{attribute 'linkalways'} 
{attribute 'no_explicit_call' := 'This FB is a CLASS and must be accessed using methods or properties'}
{attribute 'enable_dynamic_creation'}
FUNCTION_BLOCK _Array0to1_0to10OfBool EXTENDS ArrayDatatypeBase
VAR CONSTANT
	lBound : DINT := 0;
	uBound : DINT := 10;
END_VAR
VAR
	localData : ARRAY [0..1, 0..10] OF BOOL;
	activeData : REFERENCE TO ARRAY [0..1, 0..10] OF BOOL REF= localData;
	elements : ARRAY [0..1, 0..10] OF _BOOL(FALSE);
	elementLookup : Dictionary;
	baseType : _BOOL(FALSE);
END_VAR

PROPERTY PUBLIC Address : PVOID
GET
Address := ADR(activeData);
END_GET
END_PROPERTY

PROPERTY PUBLIC BaseDatatype : I_Datatype
GET
BaseDatatype := baseType;
END_GET
END_PROPERTY

METHOD PUBLIC ClearReference
VAR_INPUT
END_VAR
activeData REF= localData;
SetElementReference();
END_METHOD

METHOD PUBLIC Clone : I_Datatype
VAR
    pClone : POINTER TO _Array0to10OfBool;
END_VAR
pClone := __NEW(_Array0to10OfBool());
pClone^.Value := Value;
Clone := pClone^;
END_METHOD

METHOD FB_init : BOOL
VAR_INPUT
	bInitRetains : BOOL; // if TRUE, the retain variables are initialized (warm start / cold start)
	bInCopyCode : BOOL;  // if TRUE, the instance afterwards gets moved into the copy code (online change)
END_VAR
StoreElementsInLookup();
SetElementReference();
END_METHOD

METHOD PUBLIC GetElementAsDatatypeByIndex : I_Datatype
VAR_INPUT
	Index : DINT;
END_VAR
GetElementAsDatatypeByIndex := elements[Index];
END_METHOD

METHOD PUBLIC GetElementByIndex : REFERENCE TO _BOOL;
VAR_INPUT
	Index : DINT;
END_VAR
GetElementByIndex REF= elements[Index];
END_METHOD

PROPERTY PUBLIC LowerBound : DINT
GET
LowerBound := lBound;
END_GET
END_PROPERTY

METHOD PUBLIC MakeReferenceTo
VAR_INPUT
	ReferenceTarget : REFERENCE TO ARRAY [lBound..uBound] OF BOOL;
END_VAR
activeData REF= ReferenceTarget;
SetElementReference();
END_METHOD

METHOD PROTECTED OnSerializeArrayValues
VAR_INPUT
	Serializer : I_Serializer;
END_VAR
VAR
	i : DINT;
END_VAR
FOR i := lBound TO uBound DO
	elements[i].SerializeWith(Serializer);
END_FOR
END_METHOD

METHOD PROTECTED SetElementReference
VAR_INPUT
END_VAR
VAR
	i : DINT;
END_VAR
FOR i := lBound TO uBound DO
	elements[i].MakeReferenceTo(activeData[i]);
END_FOR
END_METHOD

PROPERTY PUBLIC Size : UDINT
GET
Size := SIZEOF(activeData);
END_GET
END_PROPERTY

METHOD PROTECTED StoreElementsInLookup
VAR_INPUT
END_VAR
FOR i := lBound TO uBound DO
	elements[i].MakeReferenceTo(activeData[i]);
END_FOR

AddElement(lookup, element[]);
END_METHOD

METHOD PROTECTED TryDeserializeArrayValues : BOOL
VAR_INPUT
	Deserializer : I_Deserializer;
	Feedback : I_DeserializerFeedback;
END_VAR
VAR
	enumerator : I_DeserializerArrayForwardEnumerator;
	i : DINT;
END_VAR
enumerator := Deserializer.GetArrayEnumerator();
i := lBound;

WHILE enumerator.MoveNext() AND i <= uBound DO
	
	IF NOT elements[i].TryDeserializeFrom(enumerator.Current, Feedback) THEN
		EXIT;
	END_IF
	i := i + 1;

END_WHILE
enumerator.Dispose();
END_METHOD

METHOD TryMakeReferenceTo : BOOL
VAR_INPUT
	Target : I_Datatype;
END_VAR
VAR
	targetAsArray : I_ArrayDatatype;
	pTargetData : POINTER TO ARRAY [lBound..uBound] OF BOOL;
END_VAR
IF NOT Target.TryResolveAsArrayDatatype(targetAsArray) THEN
	RETURN;
END_IF

IF NOT (targetAsArray.Identifier = Identifier) THEN
	RETURN;
END_IF

pTargetData := Target.Address;
activeData REF= pTargetData^;
SetElementReference();
TryMakeReferenceTo := TRUE;
END_METHOD

PROPERTY PUBLIC UpperBound : DINT
GET
UpperBound := ubound;
END_GET
END_PROPERTY

PROPERTY PUBLIC Value : REFERENCE TO ARRAY [lBound..uBound] OF BOOL;
GET
Value ref= activeData;
END_GET
END_PROPERTY

END_FUNCTION_BLOCK

(* stored: Version 1.1.0.1, ProductVersion 3.1.4024.13
   POU _Array0to1_0to10OfBool: Id {5d4a5c6c-235b-0fc8-3170-fb9e79155b24}, SpecialFunc None
   Folder Core: Id {a4c83d3b-0793-0d31-3ab4-43ec0eee571b}
   Folder Constructor: Id {f73b3dbe-bd97-0334-2b49-33e3b02f1105}
   Folder Protected: Id {f684be48-05fe-0c71-3bdd-c0a07b4c348d}
   Folder Customize: Id {51246736-122c-08bb-0d53-c36e681d4276}
   Property Address: Id {937712cb-3222-0bbc-236e-1e91efb87d64}
   Get Get: Id {7f9e12e9-d1d3-0276-13fa-4be8ae16e0f3}
   Property BaseDatatype: Id {3fe17596-775e-0ed6-18bd-5db5acebf1e5}
   Get Get: Id {5031f141-5009-0717-294e-22d89e729e2a}
   Method ClearReference: Id {a4fd45ab-9649-0f5b-046f-1eaed9fa03f4}
   Method Clone: Id {9f25814a-3a0b-04d5-3871-2c39cbe0ff34}
   Method FB_init: Id {e7c81eb0-4ae5-0991-3cb5-1f4d3b1f0247}
   Method GetElementAsDatatypeByIndex: Id {3f988d55-44c3-0ab8-22bc-a63be86b07ea}
   Method GetElementByIndex: Id {bf39b153-6231-010d-38a9-4df671a21e14}
   Property LowerBound: Id {2ae66629-81a6-0d42-0317-752dd81eb2c5}
   Get Get: Id {53ca9a66-56b4-04c9-0258-e0999a5e5328}
   Method MakeReferenceTo: Id {2fb4dcb2-2d88-0c15-3814-4a5d08cbb870}
   Method OnSerializeArrayValues: Id {4a770347-562e-0d1d-08ab-45bc07b42812}
   Method SetElementReference: Id {59c290b2-f6bb-0e03-1c68-a60a793469d4}
   Property Size: Id {b1e6b758-c1c6-0d45-1bf5-31b8e7eb4107}
   Get Get: Id {a80dcb90-cf75-06cf-04f3-df54e8e67ed9}
   Method StoreElementsInLookup: Id {bb16b1d6-082c-0f17-0145-589be290532f}
   Method TryDeserializeArrayValues: Id {3bab3720-f9eb-008c-2c4d-b192c3a7e23f}
   Method TryMakeReferenceTo: Id {ba5d49d6-2307-0f43-0db4-c34f092e36eb}
   Property UpperBound: Id {801cb29f-1364-0768-06ea-189205aadc23}
   Get Get: Id {d3e59866-b0c4-0b9c-361a-4e30ab220e06}
   Property Value: Id {579974b3-f878-0c7d-2b89-7c2e6e13bdd6}
   Get Get: Id {a0cabc49-0a70-0dce-0849-f57b718d5694} *)
